FUNCTION_BLOCK Torque EXTENDS SM_Torque
VAR_INPUT
END_VAR
VAR_OUTPUT
END_VAR
VAR
    _testVar : INT;
END_VAR

SUPER^();

END_FUNCTION_BLOCK

(* stored: Version 1.1.0.1, ProductVersion 3.1.4018.5
   POU Torque: Id {5eda0452-c252-4ade-95e5-c02bc5dcc087}, SpecialFunc None *)
